TYPE DUT_CameraReceive :
STRUCT
   iBoxType 	: INT; ;//1=锥底光滑身 2=圆底断崖身，  								 													
END_STRUCT
END_TYPE

(* stored: Version 1.1.0.1, ProductVersion 3.1.4024.9
   DUT DUT_CameraReceive: Id {20dd1f33-79c1-43f9-811a-ec321b2d7092} *)
